TYPE LoggerFirebird :
STRUCT
	MesAlarmCode		: WORD;				// Alarm Code

END_STRUCT
END_TYPE

(* stored: Version 1.1.0.1, ProductVersion 3.1.4024.6
   DUT LoggerFirebird: Id {501fc3ec-aef4-4557-a66a-125185401e9e} *)
